Fanuc KAREL source: kx00014.KL

-- PROVISIONAL review KL for V770-1; original PC SHA256 c5935904ece30845eb0028a73bd5f95d0283e069a00061f1d30b317c340c9564
-- Incomplete behavior may be omitted. Consult companion uncertainty JSON. Do not deploy.
PROGRAM KX00014
%NOLOCKGROUP
VAR
  I : INTEGER
  J : INTEGER
  B : BOOLEAN
  F : FILE
  S : STRING[80]
-- UNRESOLVED_DECL P type=000102
BEGIN
  -- UNRESOLVED_PC offsets 5-7; opcodes 9D,3C
  -- UNRESOLVED_PC offsets 12-16; opcodes 7F
END KX00014
